{attribute 'GeneratedUsingTerminal: EL2202-0100-0016'}
{attribute addProperty BoxType "EL2202-0100-0016"}
{attribute addProperty Id "Channel_1AT %Q*Channel_54BE63B32Channel_2AT %Q*Channel_54BE63B32WcStateAT %I*WcState_0B2B16F91InfoDataAT %I*InfoData_A7436BC610"}
{attribute addProperty CRC "4212322502"}
{attribute addProperty Size "15"}
TYPE EL2202_FB12F0C6 EXTENDS EtcSlaveTerminalBase_947E5A46 :
STRUCT
	{attribute addProperty Name "Channel_1"}
	Channel_1 : Channel_54BE63B3;
	{attribute addProperty Name "Channel_2"}
	Channel_2 : Channel_54BE63B3;
	{attribute addProperty Name "WcState"}
	WcState : WcState_0B2B16F9;
	{attribute addProperty Name "InfoData"}
	InfoData : InfoData_A7436BC6;
END_STRUCT
END_TYPE

(* stored: Version 1.2.0.0, ProductVersion 3.1.4024.9
   DUT EL2202_FB12F0C6: Id {2c5775e7-fda3-4207-9627-5a64e54e0d20} *)
